(* IEC 61131-3 sources: plc_simulator/services/codesys/POUs/SIM (part 2) *)

(* ---- SIM_FB_RunTasks.st ---- *)
(* ============================================================
   SIM_FB_RunTasks — Simulate transporter task execution

   Company : Galvatek part of the John Cockerill Group
   Author  : Jarmo Piipponen
   Created : 25.03.2026
   ============================================================
   For each active transporter [1..3], checks whether a new task
   has been assigned (task_id <> running_task_id) and executes
   the full transport cycle:

     Phase 0  idle        — waiting for new task
     Phase 1  to_lift     — X-drive towards lift station
     Phase 2  lifting     — Z-lift sequence (stages 1-5)
     Phase 3  to_sink     — X-drive towards sink station
     Phase 4  sinking     — Z-sink sequence (stages 6-8)

   Also maintains current_station (nearest station) every cycle.
   Called once per PLC scan from PLC_PRG.
   ------------------------------------------------------------
   Changes:
   ============================================================ *)

FUNCTION_BLOCK SIM_FB_RunTasks
VAR_INPUT
  i_run : BOOL;       (* enable — typically init_done *)
END_VAR
VAR_EXTERNAL CONSTANT
    MAX_Transporters    : INT;
    MAX_Units           : INT;
    MAX_STEPS_PER_PROGRAM          : INT;
    MIN_StationIndex : INT;
    MAX_StationIndex   : INT;
    IN_PROCESS          : INT;
END_VAR

VAR_EXTERNAL
  g_transporter  : ARRAY[1..MAX_Transporters] OF UDT_TransporterStatusType;
  g_sim_trans    : ARRAY[1..MAX_Transporters] OF UDT_JC_SimTransporterType;
  g_station     : ARRAY[MIN_StationIndex..MAX_StationIndex] OF UDT_StationType;    g_station_loc  : ARRAY[1..MAX_StationIndex] OF UDT_UnitLocation;  g_cfg          : ARRAY[1..MAX_Transporters] OF UDT_TransporterType;
  g_move         : ARRAY[1..MAX_Transporters] OF UDT_JC_MoveTimesType;
  g_actual_move  : ARRAY[1..MAX_Transporters] OF UDT_JC_ActualMoveTimeType;
  g_unit         : ARRAY[1..MAX_Units] OF UDT_UnitType;
  g_batch        : ARRAY[1..MAX_Units] OF UDT_BatchType;
  g_program      : ARRAY[1..MAX_Units] OF UDT_TreatmentProgramType;
  g_time_s       : LINT;
  g_event_pending       : UDT_JC_EventMsgType;
  g_event_pending_valid : BOOL;
END_VAR
VAR
  i            : INT;
  idx          : INT;
  (* Physics FB instances — one per transporter (MATIEC needs separate instances) *)
  fb_x1        : SIM_FB_XMotion;
  fb_x2        : SIM_FB_XMotion;
  fb_x3        : SIM_FB_XMotion;
  fb_z1        : SIM_FB_ZMotion;
  fb_z2        : SIM_FB_ZMotion;
  fb_z3        : SIM_FB_ZMotion;
  (* Station lookup — now FC SIM_FindStation, no instance needed *)
  (* Temp vars for VAR_IN_OUT passing *)
  tmp_x        : DINT;
  tmp_vx       : DINT;
  tmp_z        : DINT;
  tmp_zs       : INT;
  tmp_zt       : REAL;
  arrived_x    : BOOL;
  at_station   : BOOL;    (* TRUE only when actually at station, not just at drive limit *)
  arrived_z    : BOOL;
  station_kind : INT;
  device_delay : REAL;
  drop_time    : REAL;
  pick_unit_id : INT;     (* unit_id picked up from lift station *)
  xfer_total   : REAL;    (* transfer time for UI progress bar *)
  sink_unit_id : INT;     (* unit_id being placed at sink station *)
  (* Nearest-station calculation *)
  nearest_num  : INT;
  min_dist     : DINT;
  dx           : DINT;
  (* Actual move time tracker — now FC STC_TrackMoveTimes, no instance needed *)
  (* Unit location update — now FC STC_UpdateUnitLocation, no instance needed *)
  (* Event helpers *)
  evt_unit     : INT;
  evt_diff     : LINT;
  (* Treatment time wait *)
  can_lift       : BOOL;
  lift_uid       : INT;      (* unit at lift station *)
  treat_cal      : DINT;      (* treatment cal_time for current stage *)
  treat_elapsed  : LINT;     (* seconds spent at lift station *)
  (* ── TASK_COMPLETE event: phase timestamps per transporter ── *)
  ts_task_start  : ARRAY[1..3] OF LINT;  (* Phase 0→1: task accepted *)
  ts_at_lift     : ARRAY[1..3] OF LINT;  (* Phase 1 at_station: arrived at lift *)
  ts_lift_begin  : ARRAY[1..3] OF LINT;  (* Phase 1→2: can_lift, begin lift *)
  ts_lift_done   : ARRAY[1..3] OF LINT;  (* Phase 2→3: lift complete *)
  ts_at_sink     : ARRAY[1..3] OF LINT;  (* Phase 3→4: arrived at sink *)
  (* TASK_COMPLETE temp vars *)
  dd_lift_s      : INT;   (* lift device_delay in seconds *)
  dropping_s     : INT;   (* dropping/valutus time in seconds *)
  trip_s         : INT;   (* drip tray delay in seconds, 0 if not used *)
  dur_nosto      : INT;   (* computed nosto duration *)
  dur_lasku      : INT;   (* computed lasku duration *)
END_VAR

IF NOT i_run THEN
  RETURN;
END_IF;

FOR i := 1 TO MAX_Transporters DO
  IF g_transporter[i].IsActive THEN

  (* ── Phase 0 → 1: Accept new task ───────────────────────── *)
  IF (g_transporter[i].Phase = 0)
     AND (g_transporter[i].TaskId <> g_sim_trans[i].RunningTaskId) THEN
    g_sim_trans[i].RunningTaskId := g_transporter[i].TaskId;
    g_transporter[i].XFinalTarget := SIM_FindStation(station_number := g_transporter[i].LiftStationTarget);
    g_transporter[i].Phase := 1;
    STC_TrackMoveTimes(i_trans := i, i_prev := 0, i_new := 1);
    g_transporter[i].Status := 4;  (* auto_run *)
    g_sim_trans[i].ZStage := 0;
    g_sim_trans[i].ZTimer := 0.0;
    (* Record task start timestamp *)
    ts_task_start[i] := g_time_s;
    ts_at_lift[i]    := LINT#0;

  (* ── Phase 1: Drive X towards lift station ──────────────── *)
  ELSIF g_transporter[i].Phase = 1 THEN
    tmp_x  := g_transporter[i].XPosition;
    tmp_vx := g_sim_trans[i].XVelocity;
    IF i = 1 THEN
      fb_x1(
        delta_t  := 0.02,
        x_target := g_transporter[i].XFinalTarget,
        x_min    := g_transporter[i].XMinDriveLimit,
        x_max    := g_transporter[i].XMaxDriveLimit,
        v_max    := g_cfg[i].SpeedMax_X,
        t_acc    := g_cfg[i].Acceleration_X,
        t_dec    := g_cfg[i].Deceleration_X,
        x_pos    := tmp_x,
        v_x      := tmp_vx
      );
      arrived_x := fb_x1.arrived;
    ELSIF i = 2 THEN
      fb_x2(
        delta_t  := 0.02,
        x_target := g_transporter[i].XFinalTarget,
        x_min    := g_transporter[i].XMinDriveLimit,
        x_max    := g_transporter[i].XMaxDriveLimit,
        v_max    := g_cfg[i].SpeedMax_X,
        t_acc    := g_cfg[i].Acceleration_X,
        t_dec    := g_cfg[i].Deceleration_X,
        x_pos    := tmp_x,
        v_x      := tmp_vx
      );
      arrived_x := fb_x2.arrived;
    ELSIF i = 3 THEN
      fb_x3(
        delta_t  := 0.02,
        x_target := g_transporter[i].XFinalTarget,
        x_min    := g_transporter[i].XMinDriveLimit,
        x_max    := g_transporter[i].XMaxDriveLimit,
        v_max    := g_cfg[i].SpeedMax_X,
        t_acc    := g_cfg[i].Acceleration_X,
        t_dec    := g_cfg[i].Deceleration_X,
        x_pos    := tmp_x,
        v_x      := tmp_vx
      );
      arrived_x := fb_x3.arrived;
    END_IF;
    g_transporter[i].XPosition  := tmp_x;
    g_sim_trans[i].XVelocity := tmp_vx;

    (* Only transition when actually at station, not just at drive limit *)
    at_station := arrived_x
                  AND (ABS(g_transporter[i].XPosition - g_transporter[i].XFinalTarget) <= 6);
    IF at_station THEN
      g_transporter[i].CurrentStation := g_transporter[i].LiftStationTarget;
      (* Record arrival at lift station (first time only) *)
      IF ts_at_lift[i] = LINT#0 THEN
        ts_at_lift[i] := g_time_s;
      END_IF;

      (* ── Wait for treatment time AND device_delay before lifting ──
         Z-movement starts when the LONGER of two has elapsed:
         1. Remaining treatment time (unit must finish treatment)
         2. Station device_delay (covers must be open)
         Both timers run simultaneously from transporter arrival.
         This matches JS behavior: max(treatment, device_delay). *)
      can_lift := TRUE;
      SIM_FindStation(station_number := g_transporter[i].LiftStationTarget, device_delay_s => device_delay, dropping_time_s => drop_time);

      (* Check treatment time *)
      lift_uid := g_station_loc[g_transporter[i].LiftStationTarget].UnitId;
      IF lift_uid >= 1 AND lift_uid <= MAX_Units THEN
        IF g_batch[lift_uid].State = IN_PROCESS
           AND g_batch[lift_uid].CurStage >= 1
           AND g_batch[lift_uid].CurStage <= MAX_STEPS_PER_PROGRAM THEN
          treat_cal := g_program[lift_uid].Steps[g_batch[lift_uid].CurStage].CalTime;
          IF treat_cal > 0 THEN
            treat_elapsed := g_time_s - g_station_loc[g_transporter[i].LiftStationTarget].ChangeTime;
            IF treat_elapsed < DINT_TO_LINT(treat_cal) THEN
              can_lift := FALSE;
            END_IF;
          END_IF;
        END_IF;
      END_IF;

      (* Check device_delay — covers must have had time to open since arrival *)
      IF can_lift AND device_delay > 0.0 THEN
        IF LINT_TO_REAL(g_time_s - ts_at_lift[i]) < device_delay THEN
          can_lift := FALSE;
        END_IF;
      END_IF;

      IF can_lift THEN
      (* Record lift begin timestamp *)
      ts_lift_begin[i] := g_time_s;
      (* drop_time already captured by STC_FindStation above *)
      (* Skip stage 1 — device_delay already overlapped above.
         Z-movement starts immediately (stage 2).
         dropping_time and drip_tray_delay happen at the TOP. *)
      g_transporter[i].ZPosition := 0;
      g_sim_trans[i].ZTimer := 0.0;
      g_sim_trans[i].ZStage := 2;
      g_transporter[i].Phase := 2;
      STC_TrackMoveTimes(i_trans := i, i_prev := 1, i_new := 2);

      (* ── Calculate transfer time (used by event + batch times) ── *)
      xfer_total := STC_CalcTransferTime(
        i_from_stn            := g_transporter[i].LiftStationTarget,
        i_to_stn              := g_transporter[i].SinkStationTarget,
        i_move                := g_move[i],
        i_from_dropping_x10   := g_station[g_transporter[i].LiftStationTarget].DrippingTime,
        i_to_device_delay_x10 := g_station[g_transporter[i].SinkStationTarget].DeviceDelay,
        i_drip_tray_delay_x10 := g_cfg[i].DripTrayDelay
      );
      IF xfer_total < 1.0 THEN
        xfer_total := INT_TO_REAL(
          ABS(g_transporter[i].SinkStationTarget
              - g_transporter[i].LiftStationTarget)
        ) * 8.0;
      END_IF;
      IF xfer_total < 5.0 THEN xfer_total := 60.0; END_IF;

      (* ── Emit LIFT event (msg_type=2) ── *)
      evt_unit := g_station_loc[g_transporter[i].LiftStationTarget].UnitId;
      IF NOT g_event_pending_valid AND evt_unit >= 1 THEN
        g_event_pending.MsgType := 2;
        g_event_pending.TsHi := LINT_TO_INT(g_time_s / LINT#65536);
        g_event_pending.TsLo := LINT_TO_INT(g_time_s MOD LINT#65536);
        g_event_pending.Payload[1]  := LINT_TO_INT(g_transporter[i].TaskId / LINT#65536);   (* TaskId_Hi *)
        g_event_pending.Payload[2]  := LINT_TO_INT(g_transporter[i].TaskId MOD LINT#65536);  (* TaskId_Lo *)
        g_event_pending.Payload[3]  := i;
        g_event_pending.Payload[4]  := evt_unit;
        g_event_pending.Payload[5]  := g_transporter[i].LiftStationTarget;
        g_event_pending.Payload[6]  := g_batch[evt_unit].BatchCode;
        g_event_pending.Payload[7]  := g_batch[evt_unit].CurStage;
        evt_diff := g_time_s - g_station_loc[g_transporter[i].LiftStationTarget].ChangeTime;
        IF evt_diff > LINT#32000 THEN
          g_event_pending.Payload[8] := 32000;
        ELSE
          g_event_pending.Payload[8] := LINT_TO_INT(evt_diff);
        END_IF;
        (* ── Original program calc/min/max for this stage ── *)
        (* g_sim_trans holds dispatch-time scheduler values which may differ
           from the treatment program originals. Read directly from g_program
           using the batch's current stage (CurStage=1-based program index). *)
        IF g_batch[evt_unit].CurStage >= 1 AND g_batch[evt_unit].CurStage <= 30 THEN
          g_event_pending.Payload[9]  := DINT_TO_INT(g_program[evt_unit].Steps[g_batch[evt_unit].CurStage].CalTime);
          g_event_pending.Payload[10] := DINT_TO_INT(g_program[evt_unit].Steps[g_batch[evt_unit].CurStage].MinTime);
          g_event_pending.Payload[11] := DINT_TO_INT(g_program[evt_unit].Steps[g_batch[evt_unit].CurStage].MaxTime);
        ELSE
          (* Stage 0 (pickup) — no program step *)
          g_event_pending.Payload[9]  := 0;
          g_event_pending.Payload[10] := 0;
          g_event_pending.Payload[11] := 0;
        END_IF;
        g_event_pending.Payload[12] := REAL_TO_INT(xfer_total);
        g_event_pending_valid := TRUE;
      END_IF;

      (* Unit moves from lift station → transporter *)
      pick_unit_id := g_station_loc[g_transporter[i].LiftStationTarget].UnitId;
      IF pick_unit_id >= 1 THEN
        STC_UpdateUnitLocation(i_unit := pick_unit_id, i_location := i, i_ntt_primary := 0);

        (* Set batch transfer times for UI progress bar — matches JS behavior *)
        g_batch[pick_unit_id].StartTime := g_time_s;
        g_batch[pick_unit_id].CalTime   := REAL_TO_DINT(xfer_total);
        g_batch[pick_unit_id].MinTime   := g_batch[pick_unit_id].CalTime;
        g_batch[pick_unit_id].MaxTime   := 600;
      END_IF;
      END_IF;  (* can_lift *)
    END_IF;
    (* If arrived_x but not at_station → at drive limit, wait for clearance *)

  (* ── Phase 2: Lift Z at lift station ────────────────────── *)
  ELSIF g_transporter[i].Phase = 2 THEN
    SIM_FindStation(station_number := g_transporter[i].LiftStationTarget, skind => station_kind);
    tmp_z  := g_transporter[i].ZPosition;
    tmp_zs := g_sim_trans[i].ZStage;
    tmp_zt := g_sim_trans[i].ZTimer;
    IF i = 1 THEN
      fb_z1(
        delta_t       := 0.02,
        station_kind  := station_kind,
        ZPosDown        := g_cfg[i].ZPosDown,
        ZPosUp          := 0,
        ZPosSlowUp      := g_cfg[i].ZPosSlowUp,
        ZPosSlowDown    := g_cfg[i].ZPosSlowDown,
        ZPosSlowEnd     := g_cfg[i].ZPosSlowEnd,
        SpeedLiftSlow_Z := g_cfg[i].SpeedLiftSlow_Z,
        SpeedLiftFast_Z := g_cfg[i].SpeedLiftFast_Z,
        DripTrayDelay   := g_cfg[i].DripTrayDelay,
        DroppingTime    := g_station[g_transporter[i].LiftStationTarget].DrippingTime,
        z_mm          := tmp_z,
        z_stage       := tmp_zs,
        z_timer_s     := tmp_zt
      );
      arrived_z := fb_z1.done;
    ELSIF i = 2 THEN
      fb_z2(
        delta_t       := 0.02,
        station_kind  := station_kind,
        ZPosDown        := g_cfg[i].ZPosDown,
        ZPosUp          := 0,
        ZPosSlowUp      := g_cfg[i].ZPosSlowUp,
        ZPosSlowDown    := g_cfg[i].ZPosSlowDown,
        ZPosSlowEnd     := g_cfg[i].ZPosSlowEnd,
        SpeedLiftSlow_Z := g_cfg[i].SpeedLiftSlow_Z,
        SpeedLiftFast_Z := g_cfg[i].SpeedLiftFast_Z,
        DripTrayDelay   := g_cfg[i].DripTrayDelay,
        DroppingTime    := g_station[g_transporter[i].LiftStationTarget].DrippingTime,
        z_mm          := tmp_z,
        z_stage       := tmp_zs,
        z_timer_s     := tmp_zt
      );
      arrived_z := fb_z2.done;
    ELSIF i = 3 THEN
      fb_z3(
        delta_t       := 0.02,
        station_kind  := station_kind,
        ZPosDown        := g_cfg[i].ZPosDown,
        ZPosUp          := 0,
        ZPosSlowUp      := g_cfg[i].ZPosSlowUp,
        ZPosSlowDown    := g_cfg[i].ZPosSlowDown,
        ZPosSlowEnd     := g_cfg[i].ZPosSlowEnd,
        SpeedLiftSlow_Z := g_cfg[i].SpeedLiftSlow_Z,
        SpeedLiftFast_Z := g_cfg[i].SpeedLiftFast_Z,
        DripTrayDelay   := g_cfg[i].DripTrayDelay,
        DroppingTime    := g_station[g_transporter[i].LiftStationTarget].DrippingTime,
        z_mm          := tmp_z,
        z_stage       := tmp_zs,
        z_timer_s     := tmp_zt
      );
      arrived_z := fb_z3.done;
    END_IF;
    g_transporter[i].ZPosition      := tmp_z;
    g_sim_trans[i].ZStage   := tmp_zs;
    g_sim_trans[i].ZTimer := tmp_zt;
    IF arrived_z THEN
      (* Record lift done timestamp *)
      ts_lift_done[i] := g_time_s;
      g_transporter[i].XFinalTarget := SIM_FindStation(station_number := g_transporter[i].SinkStationTarget);
      g_transporter[i].Phase := 3;
      STC_TrackMoveTimes(i_trans := i, i_prev := 2, i_new := 3);
    END_IF;

  (* ── Phase 3: Drive X towards sink station ─────────────── *)
  ELSIF g_transporter[i].Phase = 3 THEN
    tmp_x  := g_transporter[i].XPosition;
    tmp_vx := g_sim_trans[i].XVelocity;
    IF i = 1 THEN
      fb_x1(
        delta_t  := 0.02,
        x_target := g_transporter[i].XFinalTarget,
        x_min    := g_transporter[i].XMinDriveLimit,
        x_max    := g_transporter[i].XMaxDriveLimit,
        v_max    := g_cfg[i].SpeedMax_X,
        t_acc    := g_cfg[i].Acceleration_X,
        t_dec    := g_cfg[i].Deceleration_X,
        x_pos    := tmp_x,
        v_x      := tmp_vx
      );
      arrived_x := fb_x1.arrived;
    ELSIF i = 2 THEN
      fb_x2(
        delta_t  := 0.02,
        x_target := g_transporter[i].XFinalTarget,
        x_min    := g_transporter[i].XMinDriveLimit,
        x_max    := g_transporter[i].XMaxDriveLimit,
        v_max    := g_cfg[i].SpeedMax_X,
        t_acc    := g_cfg[i].Acceleration_X,
        t_dec    := g_cfg[i].Deceleration_X,
        x_pos    := tmp_x,
        v_x      := tmp_vx
      );
      arrived_x := fb_x2.arrived;
    ELSIF i = 3 THEN
      fb_x3(
        delta_t  := 0.02,
        x_target := g_transporter[i].XFinalTarget,
        x_min    := g_transporter[i].XMinDriveLimit,
        x_max    := g_transporter[i].XMaxDriveLimit,
        v_max    := g_cfg[i].SpeedMax_X,
        t_acc    := g_cfg[i].Acceleration_X,
        t_dec    := g_cfg[i].Deceleration_X,
        x_pos    := tmp_x,
        v_x      := tmp_vx
      );
      arrived_x := fb_x3.arrived;
    END_IF;
    g_transporter[i].XPosition  := tmp_x;
    g_sim_trans[i].XVelocity := tmp_vx;

    (* Only transition when actually at station, not just at drive limit *)
    at_station := arrived_x
                  AND (ABS(g_transporter[i].XPosition - g_transporter[i].XFinalTarget) <= 6);
    IF at_station THEN
      g_transporter[i].CurrentStation := g_transporter[i].SinkStationTarget;
      (* Record arrival at sink timestamp *)
      ts_at_sink[i] := g_time_s;
      SIM_FindStation(station_number := g_transporter[i].SinkStationTarget, device_delay_s => device_delay);
      g_sim_trans[i].ZTimer := device_delay + INT_TO_REAL(g_cfg[i].DripTrayDelay) / 10.0;
      g_sim_trans[i].ZStage := 6;
      g_transporter[i].Phase := 4;
      STC_TrackMoveTimes(i_trans := i, i_prev := 3, i_new := 4);
    END_IF;
    (* If arrived_x but not at_station → at drive limit, wait for clearance *)

  (* ── Phase 4: Sink Z at sink station ───────────────────── *)
  ELSIF g_transporter[i].Phase = 4 THEN
    SIM_FindStation(station_number := g_transporter[i].SinkStationTarget, skind => station_kind);
    tmp_z  := g_transporter[i].ZPosition;
    tmp_zs := g_sim_trans[i].ZStage;
    tmp_zt := g_sim_trans[i].ZTimer;
    IF i = 1 THEN
      fb_z1(
        delta_t       := 0.02,
        station_kind  := station_kind,
        ZPosDown        := g_cfg[i].ZPosDown,
        ZPosUp          := 0,
        ZPosSlowUp      := g_cfg[i].ZPosSlowUp,
        ZPosSlowDown    := g_cfg[i].ZPosSlowDown,
        ZPosSlowEnd     := g_cfg[i].ZPosSlowEnd,
        SpeedLiftSlow_Z := g_cfg[i].SpeedLiftSlow_Z,
        SpeedLiftFast_Z := g_cfg[i].SpeedLiftFast_Z,
        DripTrayDelay   := g_cfg[i].DripTrayDelay,
        DroppingTime    := 0,
        z_mm          := tmp_z,
        z_stage       := tmp_zs,
        z_timer_s     := tmp_zt
      );
      arrived_z := fb_z1.done;
    ELSIF i = 2 THEN
      fb_z2(
        delta_t       := 0.02,
        station_kind  := station_kind,
        ZPosDown        := g_cfg[i].ZPosDown,
        ZPosUp          := 0,
        ZPosSlowUp      := g_cfg[i].ZPosSlowUp,
        ZPosSlowDown    := g_cfg[i].ZPosSlowDown,
        ZPosSlowEnd     := g_cfg[i].ZPosSlowEnd,
        SpeedLiftSlow_Z := g_cfg[i].SpeedLiftSlow_Z,
        SpeedLiftFast_Z := g_cfg[i].SpeedLiftFast_Z,
        DripTrayDelay   := g_cfg[i].DripTrayDelay,
        DroppingTime    := 0,
        z_mm          := tmp_z,
        z_stage       := tmp_zs,
        z_timer_s     := tmp_zt
      );
      arrived_z := fb_z2.done;
    ELSIF i = 3 THEN
      fb_z3(
        delta_t       := 0.02,
        station_kind  := station_kind,
        ZPosDown        := g_cfg[i].ZPosDown,
        ZPosUp          := 0,
        ZPosSlowUp      := g_cfg[i].ZPosSlowUp,
        ZPosSlowDown    := g_cfg[i].ZPosSlowDown,
        ZPosSlowEnd     := g_cfg[i].ZPosSlowEnd,
        SpeedLiftSlow_Z := g_cfg[i].SpeedLiftSlow_Z,
        SpeedLiftFast_Z := g_cfg[i].SpeedLiftFast_Z,
        DripTrayDelay   := g_cfg[i].DripTrayDelay,
        DroppingTime    := 0,
        z_mm          := tmp_z,
        z_stage       := tmp_zs,
        z_timer_s     := tmp_zt
      );
      arrived_z := fb_z3.done;
    END_IF;
    g_transporter[i].ZPosition      := tmp_z;
    g_sim_trans[i].ZStage   := tmp_zs;
    g_sim_trans[i].ZTimer := tmp_zt;
    IF arrived_z THEN
      (* ── Emit TASK_COMPLETE event (msg_type=3) before Phase reset ── *)
      IF NOT g_event_pending_valid THEN
        (* Config-based sub-phase durations *)
        dropping_s := g_transporter[i].DrippingTime / 10;
        IF g_cfg[i].DripTrayInUse THEN
          trip_s := g_cfg[i].DripTrayDelay / 10;
        ELSE
          trip_s := 0;
        END_IF;
        (* Nosto = total lift phase - dropping - trip_close
           device_delay no longer in lift phase (overlapped in Phase 1) *)
        dur_nosto := LINT_TO_INT(ts_lift_done[i] - ts_lift_begin[i])
                     - dropping_s - trip_s;
        IF dur_nosto < 0 THEN dur_nosto := 0; END_IF;
        (* Lasku = total sink phase - device_delay - trip_open *)
        dd_lift_s := g_sim_trans[i].SinkDeviceDelay / 10;
        dur_lasku := LINT_TO_INT(g_time_s - ts_at_sink[i]) - dd_lift_s - trip_s;
        IF dur_lasku < 0 THEN dur_lasku := 0; END_IF;

        g_event_pending.MsgType := 3;
        g_event_pending.TsHi := LINT_TO_INT(g_time_s / LINT#65536);
        g_event_pending.TsLo := LINT_TO_INT(g_time_s MOD LINT#65536);
        g_event_pending.Payload[1]  := LINT_TO_INT(g_transporter[i].TaskId / LINT#65536);   (* TaskId_Hi *)
        g_event_pending.Payload[2]  := LINT_TO_INT(g_transporter[i].TaskId MOD LINT#65536);  (* TaskId_Lo *)
        g_event_pending.Payload[3]  := i;                                                     (* transporter *)
        g_event_pending.Payload[4]  := LINT_TO_INT(ts_at_lift[i] - ts_task_start[i]);         (* siirto nostoasemalle *)
        g_event_pending.Payload[5]  := LINT_TO_INT(ts_lift_begin[i] - ts_at_lift[i]);         (* odotus ennen nostoa (max(treat,dev_delay)) *)
        g_event_pending.Payload[6]  := dur_nosto;                                             (* nosto *)
        g_event_pending.Payload[7]  := dropping_s;                                            (* valutus *)
        g_event_pending.Payload[8]  := trip_s;                                                (* trip close *)
        g_event_pending.Payload[9]  := LINT_TO_INT(ts_at_sink[i] - ts_lift_done[i]);          (* siirto laskuasemalle *)
        g_event_pending.Payload[10] := trip_s;                                                (* trip open *)
        g_event_pending.Payload[11] := dur_lasku;                                             (* lasku *)
        g_event_pending.Payload[12] := LINT_TO_INT(g_time_s - ts_task_start[i]);              (* total *)
        g_event_pending_valid := TRUE;
      END_IF;

      (* Unit moves from transporter → sink station *)
      sink_unit_id := g_station_loc[i].UnitId;
      IF sink_unit_id >= 1 THEN
        STC_UpdateUnitLocation(i_unit := sink_unit_id, i_location := g_transporter[i].SinkStationTarget, i_ntt_primary := g_sim_trans[i].NttPrimary);
      END_IF;

      g_transporter[i].Phase := 0;
      STC_TrackMoveTimes(i_trans := i, i_prev := 4, i_new := 0);
      g_transporter[i].Status := 3;  (* auto_idle *)

    END_IF;
  END_IF;  (* ELSIF chain: phases 0→1→2→3→4 *)

  (* ── Phase 0 idle: drive back inside limits if outside ────── *)
  IF g_transporter[i].Phase = 0 THEN
    tmp_x  := g_transporter[i].XPosition;
    tmp_vx := g_sim_trans[i].XVelocity;
    (* Use current position as target — XMotion will clamp to nearest limit if outside *)
    IF i = 1 THEN
      fb_x1(
        delta_t  := 0.02,
        x_target := tmp_x,
        x_min    := g_transporter[i].XMinDriveLimit,
        x_max    := g_transporter[i].XMaxDriveLimit,
        v_max    := g_cfg[i].SpeedMax_X,
        t_acc    := g_cfg[i].Acceleration_X,
        t_dec    := g_cfg[i].Deceleration_X,
        x_pos    := tmp_x,
        v_x      := tmp_vx
      );
    ELSIF i = 2 THEN
      fb_x2(
        delta_t  := 0.02,
        x_target := tmp_x,
        x_min    := g_transporter[i].XMinDriveLimit,
        x_max    := g_transporter[i].XMaxDriveLimit,
        v_max    := g_cfg[i].SpeedMax_X,
        t_acc    := g_cfg[i].Acceleration_X,
        t_dec    := g_cfg[i].Deceleration_X,
        x_pos    := tmp_x,
        v_x      := tmp_vx
      );
    ELSIF i = 3 THEN
      fb_x3(
        delta_t  := 0.02,
        x_target := tmp_x,
        x_min    := g_transporter[i].XMinDriveLimit,
        x_max    := g_transporter[i].XMaxDriveLimit,
        v_max    := g_cfg[i].SpeedMax_X,
        t_acc    := g_cfg[i].Acceleration_X,
        t_dec    := g_cfg[i].Deceleration_X,
        x_pos    := tmp_x,
        v_x      := tmp_vx
      );
    END_IF;
    g_transporter[i].XPosition  := tmp_x;
    g_sim_trans[i].XVelocity := tmp_vx;
  END_IF;

  (* ── Nearest station tracking ──────────────────────────── *)
  min_dist := 999999999;
  nearest_num := g_transporter[i].CurrentStation;
  FOR idx := MIN_StationIndex TO MAX_StationIndex DO
    IF g_station[idx].TankId <> 0 THEN
      dx := g_station[idx].XPosition - g_transporter[i].XPosition;
      IF ABS(dx) < min_dist THEN
        min_dist := ABS(dx);
        nearest_num := idx;
      END_IF;
    END_IF;
  END_FOR;
  g_transporter[i].CurrentStation := nearest_num;

  END_IF;  (* active *)
END_FOR;

END_FUNCTION_BLOCK

(* ---- SIM_FB_XMotion.st ---- *)
(* ============================================================
   SIM_FB_XMotion — Horizontal motion with accel / decel

   Company : Galvatek part of the John Cockerill Group
   Author  : Jarmo Piipponen
   Created : 25.03.2026
   ============================================================
   Trapezoidal velocity profile: accelerate, cruise, decelerate.
   Clamps position to [x_min..x_max] drive limits.
   VAR_IN_OUT: x_pos, v_x (modified in place).
   ------------------------------------------------------------
   Changes:
   ============================================================ *)

FUNCTION_BLOCK SIM_FB_XMotion
VAR_INPUT
  delta_t  : REAL;     (* cycle time s — simulation internal *)
  x_target : DINT;     (* target X mm *)
  x_min    : DINT;     (* TWA lower limit mm *)
  x_max    : DINT;     (* TWA upper limit mm *)
  v_max    : DINT;     (* max velocity mm/s *)
  t_acc    : DINT;     (* acceleration time ×10 = tenths of second *)
  t_dec    : DINT;     (* deceleration time ×10 = tenths of second *)
END_VAR
VAR_IN_OUT
  x_pos : DINT;        (* current X position mm *)
  v_x   : DINT;        (* current X velocity mm/s *)
END_VAR
VAR_OUTPUT
  arrived : BOOL;
  x_drive : DINT;      (* actual drive target after limit clamping *)
END_VAR
VAR
  (* Internal REAL copies for physics integration *)
  r_target     : REAL;
  r_min        : REAL;
  r_max        : REAL;
  r_vmax       : REAL;
  r_tacc       : REAL;
  r_tdec       : REAL;
  r_pos        : REAL;
  r_vel        : REAL;
  drive_target : REAL;
  distance     : REAL;
  dir          : REAL;
  a_acc        : REAL;
  a_dec        : REAL;
  brake_dist   : REAL;
  new_vel      : REAL;
  travel       : REAL;
END_VAR
  (* Convert DINT/INT inputs to REAL for physics *)
  r_target := DINT_TO_REAL(x_target);
  r_min    := DINT_TO_REAL(x_min);
  r_max    := DINT_TO_REAL(x_max);
  r_vmax   := DINT_TO_REAL(v_max);
  r_tacc   := DINT_TO_REAL(t_acc) / 10.0;
  r_tdec   := DINT_TO_REAL(t_dec) / 10.0;
  r_pos    := DINT_TO_REAL(x_pos);
  r_vel    := DINT_TO_REAL(v_x);

  IF (r_max > r_min) THEN
    IF r_pos < r_min THEN
      drive_target := r_min;
    ELSIF r_pos > r_max THEN
      drive_target := r_max;
    ELSE
      IF r_target < r_min THEN
        drive_target := r_min;
      ELSIF r_target > r_max THEN
        drive_target := r_max;
      ELSE
        drive_target := r_target;
      END_IF;
    END_IF;
  ELSE
    drive_target := r_target;
  END_IF;

  x_drive := REAL_TO_DINT(drive_target);

  arrived := ABS(r_pos - drive_target) <= 3.0;
  IF arrived THEN
    x_pos := REAL_TO_DINT(drive_target);
    v_x := 0;
    RETURN;
  END_IF;

  IF r_tacc <= 0.0 THEN r_tacc := 0.001; END_IF;
  IF r_tdec <= 0.0 THEN r_tdec := 0.001; END_IF;
  IF r_vmax < 0.0 THEN r_vmax := 0.0; END_IF;

  a_acc := r_vmax / r_tacc;
  a_dec := r_vmax / r_tdec;

  dir := 1.0;
  IF drive_target < r_pos THEN
    dir := -1.0;
  END_IF;

  distance := ABS(drive_target - r_pos);

  IF a_dec > 0.0 THEN
    brake_dist := (r_vel * r_vel) / (2.0 * a_dec);
  ELSE
    brake_dist := 0.0;
  END_IF;

  IF brake_dist >= distance THEN
    new_vel := r_vel - a_dec * delta_t;
    IF new_vel < 0.0 THEN new_vel := 0.0; END_IF;
  ELSE
    new_vel := r_vel + a_acc * delta_t;
    IF new_vel > r_vmax THEN new_vel := r_vmax; END_IF;
  END_IF;

  travel := new_vel * delta_t;
  IF travel >= distance THEN
    x_pos := REAL_TO_DINT(drive_target);
    v_x := 0;
    arrived := TRUE;
  ELSE
    x_pos := REAL_TO_DINT(r_pos + dir * travel);
    v_x := REAL_TO_DINT(new_vel);
    arrived := FALSE;
  END_IF;
END_FUNCTION_BLOCK

(* ---- SIM_FB_ZMotion.st ---- *)
(* ============================================================
   SIM_FB_ZMotion — Vertical (Z) motion simulation

   Company : Galvatek part of the John Cockerill Group
   Author  : Jarmo Piipponen
   Created : 25.03.2026
   ============================================================
   Simulates 2D transporter lift/sink with realistic physics:
   slow start / fast middle / slow end speed profiles,
   different slow zones for wet vs dry stations.

   LIFT sequence (z_stage 2-5, 9):
     2: Slow lift    0 → ZPosSlowUp/ZPosSlowDown
     3: Fast lift    → (z_total - ZPosSlowEnd)
     4: Slow end     → z_total
     5: Dropping     at top, dripping time
     9: Drip close   drip tray close delay at top

   SINK sequence (z_stage 6-8):
     6: Init delay   (device_delay + drip_delay)
     7: Fast sink    z_total → slow_zone
     8: Slow sink    → 0 mm

   Caller sets z_stage and z_timer_s before first call.
   Output 'done' pulses TRUE when sequence completes.
   ------------------------------------------------------------
   Changes:
   ============================================================ *)

FUNCTION_BLOCK SIM_FB_ZMotion
VAR_INPUT
  delta_t         : REAL;    (* Cycle time in seconds — simulation internal *)
  station_kind    : INT;     (* KIND_DRY=0, KIND_WET=1 *)
  ZPosUp          : DINT;    (* Z position at full up mm *)
  ZPosDown        : DINT;    (* Z position at full down mm *)
  ZPosSlowUp      : DINT;    (* Slow zone when going up (dry) mm *)
  ZPosSlowDown    : DINT;    (* Slow zone when going down (wet) mm *)
  ZPosSlowEnd     : DINT;    (* Slow zone at end of travel mm *)
  SpeedLiftSlow_Z : DINT;    (* Slow speed mm/s *)
  SpeedLiftFast_Z : DINT;    (* Fast speed mm/s *)
  DripTrayDelay   : INT;     (* Drip tray open/close delay ×10 = tenths of second *)
  DroppingTime    : INT;     (* Dropping/dripping time ×10 = tenths of second *)
END_VAR
VAR_IN_OUT
  z_mm      : DINT;        (* Current Z position mm *)
  z_stage   : INT;         (* Current motion stage *)
  z_timer_s : REAL;        (* Delay timer — simulation internal *)
END_VAR
VAR_OUTPUT
  done : BOOL;             (* TRUE when sequence complete *)
END_VAR
VAR_EXTERNAL CONSTANT
  KIND_WET : INT;
END_VAR
VAR
  (* Internal REAL copies for physics integration *)
  r_z          : REAL;
  r_total      : REAL;
  r_slow_zone  : REAL;
  r_slow_end   : REAL;
  r_slow_spd   : REAL;
  r_fast_spd   : REAL;
  r_drip       : REAL;
  r_drop       : REAL;     (* dropping/dripping time seconds *)
  z_total_mm   : DINT;     (* computed: ZPosDown - ZPosUp *)
END_VAR

  done := FALSE;
  z_total_mm := ZPosDown - ZPosUp;

  (* Convert DINT/INT inputs to REAL for physics *)
  r_z         := DINT_TO_REAL(z_mm);
  r_total     := DINT_TO_REAL(z_total_mm);
  r_slow_end  := DINT_TO_REAL(ZPosSlowEnd);
  r_slow_spd  := DINT_TO_REAL(SpeedLiftSlow_Z);
  r_fast_spd  := DINT_TO_REAL(SpeedLiftFast_Z);
  r_drip      := INT_TO_REAL(DripTrayDelay) / 10.0;
  r_drop      := INT_TO_REAL(DroppingTime) / 10.0;

  (* Select slow zone based on station kind *)
  IF station_kind = KIND_WET THEN
    r_slow_zone := DINT_TO_REAL(ZPosSlowDown);
  ELSE
    r_slow_zone := DINT_TO_REAL(ZPosSlowUp);
  END_IF;

  CASE z_stage OF

    (* === LIFT: stages 2-5,9 — nosto altaasta ylös (z kasvaa: 0 → z_total) === *)
    (* Stage 1 no longer used for lift — device_delay overlaps with treatment wait *)

    2: (* Slow lift start — hidas nosto nesteestä *)
      r_z := r_z + r_slow_spd * delta_t;
      z_mm := REAL_TO_DINT(r_z);
      IF r_z >= r_slow_zone THEN
        z_stage := 3;
      END_IF;

    3: (* Fast lift — nopea nosto *)
      r_z := r_z + r_fast_spd * delta_t;
      z_mm := REAL_TO_DINT(r_z);
      IF r_z >= (r_total - r_slow_end) THEN
        z_stage := 4;
      END_IF;

    4: (* Slow lift end — hidas loppunosto *)
      r_z := r_z + r_slow_spd * delta_t;
      IF r_z >= r_total THEN
        z_mm := z_total_mm;
        z_timer_s := r_drop;
        z_stage := 5;
      ELSE
        z_mm := REAL_TO_DINT(r_z);
      END_IF;

    5: (* Dropping / dripping — valutusaika yläasemassa *)
      z_timer_s := z_timer_s - delta_t;
      IF z_timer_s <= 0.0 THEN
        z_timer_s := r_drip;
        z_stage := 9;
      END_IF;

    9: (* Drip tray close — tippakouru sulkeutuu *)
      z_timer_s := z_timer_s - delta_t;
      IF z_timer_s <= 0.0 THEN
        z_stage := 0;
        done := TRUE;
      END_IF;

    (* === SINK: stages 6-8 — lasku altaaseen (z pienenee: z_total → 0) === *)

    6: (* Init delay: device_delay + drip_delay *)
      z_timer_s := z_timer_s - delta_t;
      IF z_timer_s <= 0.0 THEN
        z_stage := 7;
      END_IF;

    7: (* Fast sink — nopea lasku *)
      r_z := r_z - r_fast_spd * delta_t;
      z_mm := REAL_TO_DINT(r_z);
      IF r_z <= r_slow_zone THEN
        z_stage := 8;
      END_IF;

    8: (* Slow sink — hidas lasku nesteeseen *)
      r_z := r_z - r_slow_spd * delta_t;
      IF r_z <= 0.0 THEN
        z_mm := 0;
        z_stage := 0;
        done := TRUE;
      ELSE
        z_mm := REAL_TO_DINT(r_z);
      END_IF;

  END_CASE;

END_FUNCTION_BLOCK
